// Mitsubishi GX Works2 project: Project   PLC: FX3U/FX3UC

PROGRAM MAIN
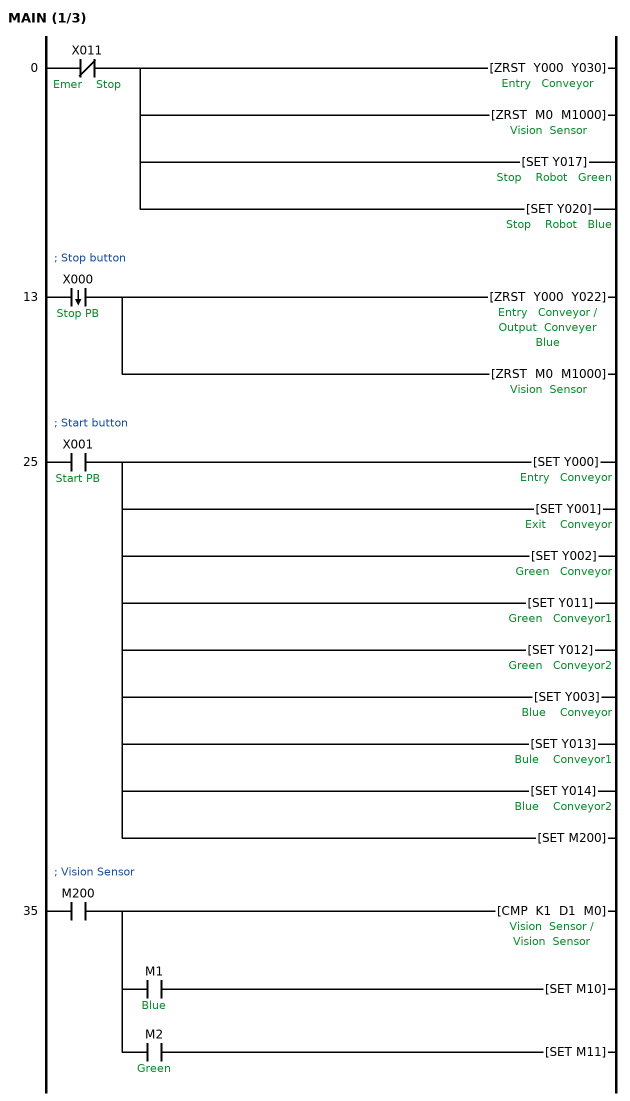
0     LDI     X011  ; Emer    Stop
      ZRST    Y000 Y030  ; Entry   Conveyor
      ZRST    M0 M1000  ; Vision  Sensor
      SET     Y017  ; Stop    Robot   Green
      SET     Y020  ; Stop    Robot   Blue
; Stop button
13    LDF     X000  ; Stop PB
      ZRST    Y000 Y022  ; Output  ConveyerBlue
      ZRST    M0 M1000
; Start button
25    LD      X001  ; Start PB
      SET     Y000  ; Entry   Conveyor
      SET     Y001  ; Exit    Conveyor
      SET     Y002  ; Green   Conveyor
      SET     Y011  ; Green   Conveyor1
      SET     Y012  ; Green   Conveyor2
      SET     Y003  ; Blue    Conveyor
      SET     Y013  ; Bule    Conveyor1
      SET     Y014  ; Blue    Conveyor2
      SET     M200
; Vision Sensor
35    LD      M200
      CMP     K1 D1 M0  ; Vision  Sensor
      MPS
      AND     M1  ; Blue
      SET     M10
      MPP
      AND     M2  ; Green
      SET     M11
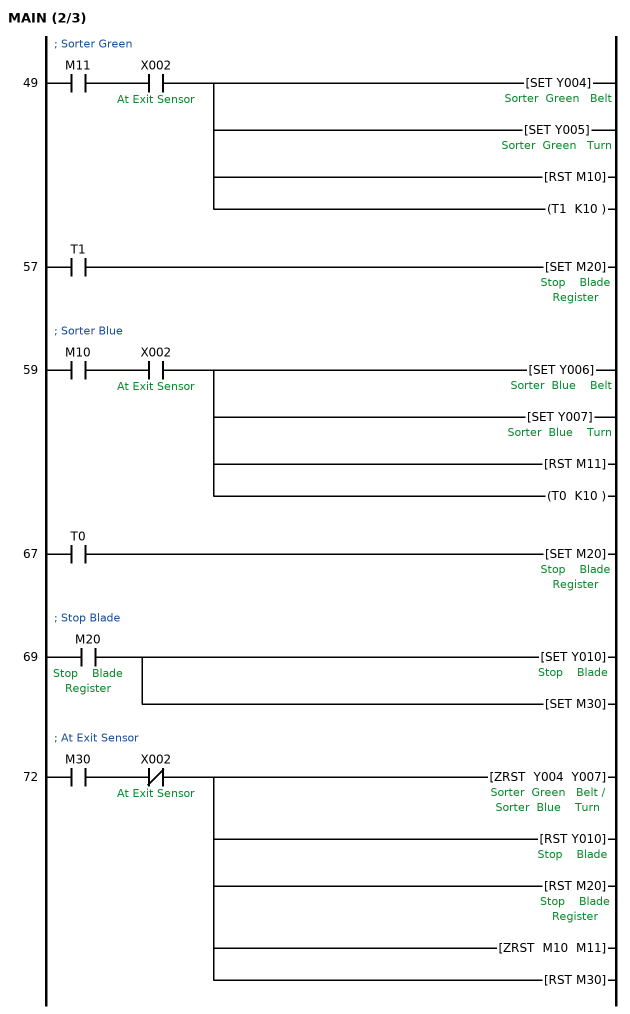
; Sorter Green
49    LD      M11
      AND     X002  ; At Exit Sensor
      SET     Y004  ; Sorter  Green   Belt
      SET     Y005  ; Sorter  Green   Turn
      RST     M10
      OUT     T1 K10
57    LD      T1
      SET     M20  ; Stop    Blade   Register
; Sorter Blue
59    LD      M10
      AND     X002  ; At Exit Sensor
      SET     Y006  ; Sorter  Blue    Belt
      SET     Y007  ; Sorter  Blue    Turn
      RST     M11
      OUT     T0 K10
67    LD      T0
      SET     M20  ; Stop    Blade   Register
; Stop Blade
69    LD      M20  ; Stop    Blade   Register
      SET     Y010  ; Stop    Blade
      SET     M30
; At Exit Sensor
72    LD      M30
      ANI     X002  ; At Exit Sensor
      ZRST    Y004 Y007
      RST     Y010  ; Stop    Blade
      RST     M20  ; Stop    Blade   Register
      ZRST    M10 M11
      RST     M30
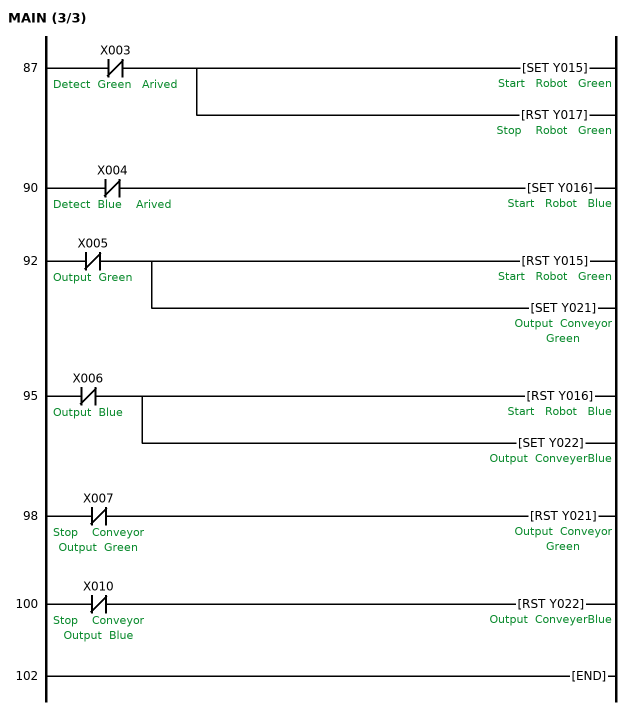
87    LDI     X003  ; Detect  Green   Arived
      SET     Y015  ; Start   Robot   Green
      RST     Y017  ; Stop    Robot   Green
90    LDI     X004  ; Detect  Blue    Arived
      SET     Y016  ; Start   Robot   Blue
92    LDI     X005  ; Output  Green
      RST     Y015  ; Start   Robot   Green
      SET     Y021  ; Output  ConveyorGreen
95    LDI     X006  ; Output  Blue
      RST     Y016  ; Start   Robot   Blue
      SET     Y022  ; Output  ConveyerBlue
98    LDI     X007  ; Stop    ConveyorOutput  Green
      RST     Y021  ; Output  ConveyorGreen
100   LDI     X010  ; Stop    ConveyorOutput  Blue
      RST     Y022  ; Output  ConveyerBlue
102   END
END_PROGRAM

// device comments not shown above
M3  ; Metal
